// TIA Portal project "Handlings7300ip" (V15.1)

(* hardware
DEVICE "S7300/ET200M station_1"  S7-300 station
   slot 0: "Rail_0"  Rail  6ES7 390-1***0-0AA0
   slot 2: "PLC_1"  CPU 314C-2 PN/DP  6ES7 314-6EH04-0AB0  V3.3
      slot 2: "PROFINET interface_1"  PN-IO
         slot 1: "Port_1"  Port
         slot 2: "Port_2"  Port
      slot 5: "DI 24/DO 16_1"  DI24/DO16
      slot 6: "AI 5/AO 2_1"  AI5/AO2
      slot 7: "Count_1"  Counter
      slot 8: "Positioning_1"  Positioning
   slot 4: "DO 8x24VDC/0.5A_1"  DO8 x 24VDC / 0.5A  6ES7 322-8BF00-0AB0
*)

// ===== PLC "PLC_1"  CPU 314C-2 PN/DP =====

VAR_GLOBAL   // PLC tag table "Default tag table"
   "Auto" AT %I0.0 : Bool;
   "Manua" AT %I0.1 : Bool;
   "S1_Nipper_out" AT %I0.2 : Bool;
   "S2_Nipper_in" AT %I0.3 : Bool;
   "S3_Nipper_off" AT %I0.4 : Bool;
   "S5_Nipper_up" AT %I0.5 : Bool;
   "S6_Nipper_down" AT %I0.6 : Bool;
   "Start" AT %I1.0 : Bool;
   "Stop" AT %I1.1 : Bool;
   "Reset" AT %I1.2 : Bool;
   "A1" AT %I1.3 : Bool;
   "A2" AT %I1.4 : Bool;
   "B1" AT %I1.5 : Bool;
   "B2" AT %I2.0 : Bool;
   "C1" AT %I2.1 : Bool;
   "C2" AT %I2.2 : Bool;
   "1Y2" AT %Q0.0 : Bool;
   "1Y1" AT %Q0.1 : Bool;
   "2Y1" AT %Q0.2 : Bool;
   "M+" AT %Q0.3 : Bool;
   "M-" AT %Q0.4 : Bool;
   "H_Auto" AT %Q0.5 : Bool;
   "H_Manual" AT %Q0.6 : Bool;
END_VAR

DATA_BLOCK "Master_DB"   // DB1
{ S7_Optimized_Access := 'FALSE' }
VERSION : 0.1
// stored: InstanceOfName Master
"Master"
BEGIN
END_DATA_BLOCK

DATA_BLOCK "Auto_Mode_DB"   // DB2
{ S7_Optimized_Access := 'FALSE' }
VERSION : 0.1
// stored: InstanceOfName Auto_Mode
"Auto_Mode"
BEGIN
END_DATA_BLOCK

DATA_BLOCK "Output_DB"   // DB3
{ S7_Optimized_Access := 'FALSE' }
VERSION : 0.1
// stored: InstanceOfName Output
"Output"
BEGIN
END_DATA_BLOCK

DATA_BLOCK "Manual_Mode_DB"   // DB4
{ S7_Optimized_Access := 'FALSE' }
VERSION : 0.1
// stored: InstanceOfName Manual_Mode
"Manual_Mode"
BEGIN
END_DATA_BLOCK

DATA_BLOCK "Resets_DB"   // DB5
{ S7_Optimized_Access := 'FALSE' }
VERSION : 0.1
// stored: InstanceOfName Resets
"Resets"
BEGIN
END_DATA_BLOCK

FUNCTION_BLOCK "Master"   // FB1, FBD
{ S7_Optimized_Access := 'FALSE' }
VERSION : 0.1
   VAR_INPUT
      Auto : Bool;
      Manual : Bool;
      Start : Bool;
      Stop : Bool;
      Reset : Bool;
      S1 : Bool;
      S2 : Bool;
      S3 : Bool;
      S5 : Bool;
      S6 : Bool;
      "G_Reset.X200" : Bool;
      "G_Reset.X201" : Bool;
   END_VAR
   VAR_OUTPUT
      H_Auto : Bool;
      H_Manual : Bool;
      G_Auto_mode : Bool;
      G_Manual_mode : Bool;
   END_VAR
   VAR
      X0 : Bool;
      X1 : Bool;
      X2 : Bool;
      X3 : Bool;
   END_VAR
BEGIN

REGION Network 1
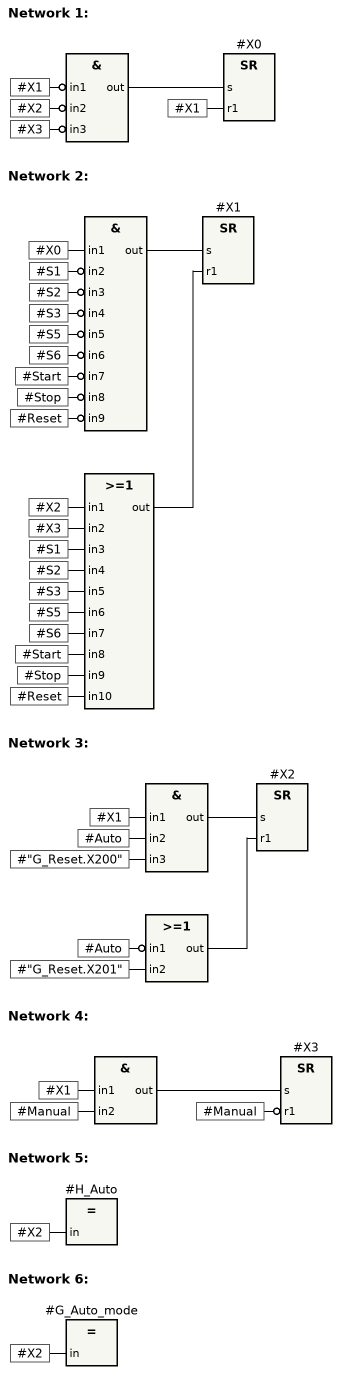
   IF NOT #X1 AND NOT #X2 AND NOT #X3 THEN
       #X0 := TRUE;   // SR flip-flop
   END_IF;
   IF #X1 THEN #X0 := FALSE; END_IF;
END_REGION

REGION Network 2
   IF #X0 AND NOT #S1 AND NOT #S2 AND NOT #S3 AND NOT #S5 AND NOT #S6 AND NOT #Start AND NOT #Stop AND NOT #Reset THEN
       #X1 := TRUE;   // SR flip-flop
   END_IF;
   IF #X2 OR #X3 OR #S1 OR #S2 OR #S3 OR #S5 OR #S6 OR #Start OR #Stop OR #Reset THEN #X1 := FALSE; END_IF;
END_REGION

REGION Network 3
   IF #X1 AND #Auto AND #"G_Reset.X200" THEN
       #X2 := TRUE;   // SR flip-flop
   END_IF;
   IF NOT #Auto OR #"G_Reset.X201" THEN #X2 := FALSE; END_IF;
END_REGION

REGION Network 4
   IF #X1 AND #Manual THEN
       #X3 := TRUE;   // SR flip-flop
   END_IF;
   IF NOT #Manual THEN #X3 := FALSE; END_IF;
END_REGION

REGION Network 5
   #H_Auto := #X2;
END_REGION

REGION Network 6
   #G_Auto_mode := #X2;
END_REGION

REGION Network 7
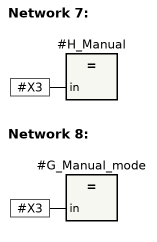
   #H_Manual := #X3;
END_REGION

REGION Network 8
   #G_Manual_mode := #X3;
END_REGION
END_FUNCTION_BLOCK

FUNCTION_BLOCK "Auto_Mode"   // FB2, FBD
{ S7_Optimized_Access := 'FALSE' }
VERSION : 0.1
   VAR_INPUT
      Auto_mode : Bool;
      Start : Bool;
      Stop : Bool;
      Reset : Bool;
      A1 : Bool;
      A2 : Bool;
      B1 : Bool;
      B2 : Bool;
      C1 : Bool;
      C2 : Bool;
   END_VAR
   VAR_OUTPUT
      Nipper_out_1Y1_A : Bool;
      Nipper_in_1Y2_A : Bool;
      Nipper_off_2Y1_A : Bool;
      Nipper_up_A : Bool;
      Nipper_down_A : Bool;
   END_VAR
   VAR
      X10 : Bool;
      X11 : Bool;
      X12 : Bool;
      X13 : Bool;
      X14 : Bool;
      X15 : Bool;
      X16 : Bool;
      X17 : Bool;
      X18 : Bool;
   END_VAR
BEGIN

REGION Network 1
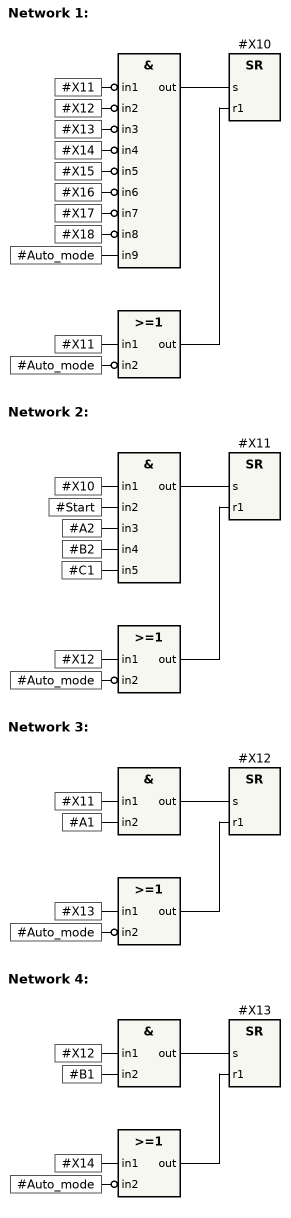
   IF NOT #X11 AND NOT #X12 AND NOT #X13 AND NOT #X14 AND NOT #X15 AND NOT #X16 AND NOT #X17 AND NOT #X18 AND #Auto_mode THEN
       #X10 := TRUE;   // SR flip-flop
   END_IF;
   IF #X11 OR NOT #Auto_mode THEN #X10 := FALSE; END_IF;
END_REGION

REGION Network 2
   IF #X10 AND #Start AND #A2 AND #B2 AND #C1 THEN
       #X11 := TRUE;   // SR flip-flop
   END_IF;
   IF #X12 OR NOT #Auto_mode THEN #X11 := FALSE; END_IF;
END_REGION

REGION Network 3
   IF #X11 AND #A1 THEN
       #X12 := TRUE;   // SR flip-flop
   END_IF;
   IF #X13 OR NOT #Auto_mode THEN #X12 := FALSE; END_IF;
END_REGION

REGION Network 4
   IF #X12 AND #B1 THEN
       #X13 := TRUE;   // SR flip-flop
   END_IF;
   IF #X14 OR NOT #Auto_mode THEN #X13 := FALSE; END_IF;
END_REGION

REGION Network 5
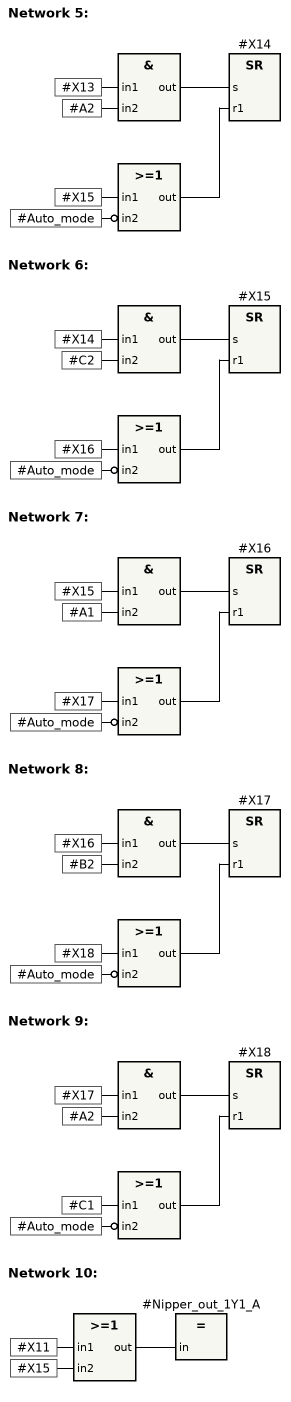
   IF #X13 AND #A2 THEN
       #X14 := TRUE;   // SR flip-flop
   END_IF;
   IF #X15 OR NOT #Auto_mode THEN #X14 := FALSE; END_IF;
END_REGION

REGION Network 6
   IF #X14 AND #C2 THEN
       #X15 := TRUE;   // SR flip-flop
   END_IF;
   IF #X16 OR NOT #Auto_mode THEN #X15 := FALSE; END_IF;
END_REGION

REGION Network 7
   IF #X15 AND #A1 THEN
       #X16 := TRUE;   // SR flip-flop
   END_IF;
   IF #X17 OR NOT #Auto_mode THEN #X16 := FALSE; END_IF;
END_REGION

REGION Network 8
   IF #X16 AND #B2 THEN
       #X17 := TRUE;   // SR flip-flop
   END_IF;
   IF #X18 OR NOT #Auto_mode THEN #X17 := FALSE; END_IF;
END_REGION

REGION Network 9
   IF #X17 AND #A2 THEN
       #X18 := TRUE;   // SR flip-flop
   END_IF;
   IF #C1 OR NOT #Auto_mode THEN #X18 := FALSE; END_IF;
END_REGION

REGION Network 10
   #Nipper_out_1Y1_A := #X11 OR #X15;
END_REGION

REGION Network 11
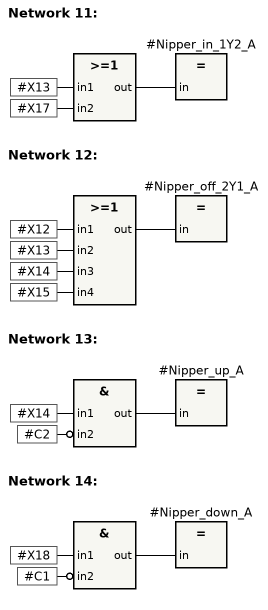
   #Nipper_in_1Y2_A := #X13 OR #X17;
END_REGION

REGION Network 12
   #Nipper_off_2Y1_A := #X12 OR #X13 OR #X14 OR #X15;
END_REGION

REGION Network 13
   #Nipper_up_A := #X14 AND NOT #C2;
END_REGION

REGION Network 14
   #Nipper_down_A := #X18 AND NOT #C1;
END_REGION
END_FUNCTION_BLOCK

FUNCTION_BLOCK "Output"   // FB3, FBD
{ S7_Optimized_Access := 'FALSE' }
VERSION : 0.1
   VAR_INPUT
      Nipper_out_1Y1_M : Bool;
      Nipper_in_1Y2_M : Bool;
      Nipper_off_2Y1_M : Bool;
      Nipper_up_M : Bool;
      Nipper_down_M : Bool;
      Nipper_out_1Y1_A : Bool;
      Nipper_in_1Y2_A : Bool;
      Nipper_off_2Y1_A : Bool;
      Nipper_up_A : Bool;
      Nipper_down_A : Bool;
      Nipper_in_1Y2_r : Bool;
      Nipper_off_2Y1_r : Bool;
      Nipper_down_r : Bool;
   END_VAR
   VAR_OUTPUT
      Nipper_out_1Y1 : Bool;
      Nipper_in_1Y2 : Bool;
      Nipper_off_2Y1 : Bool;
      Nipper_up : Bool;
      Nipper_down : Bool;
   END_VAR
BEGIN

REGION Network 1
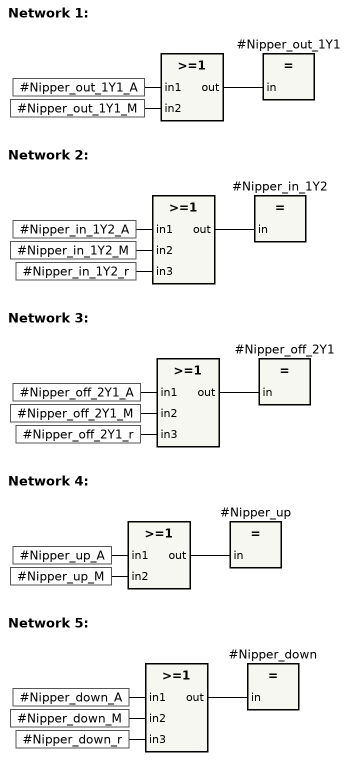
   #Nipper_out_1Y1 := #Nipper_out_1Y1_A OR #Nipper_out_1Y1_M;
END_REGION

REGION Network 2
   #Nipper_in_1Y2 := #Nipper_in_1Y2_A OR #Nipper_in_1Y2_M OR #Nipper_in_1Y2_r;
END_REGION

REGION Network 3
   #Nipper_off_2Y1 := #Nipper_off_2Y1_A OR #Nipper_off_2Y1_M OR #Nipper_off_2Y1_r;
END_REGION

REGION Network 4
   #Nipper_up := #Nipper_up_A OR #Nipper_up_M;
END_REGION

REGION Network 5
   #Nipper_down := #Nipper_down_A OR #Nipper_down_M OR #Nipper_down_r;
END_REGION
END_FUNCTION_BLOCK

FUNCTION_BLOCK "Manual_Mode"   // FB4, FBD
{ S7_Optimized_Access := 'FALSE' }
VERSION : 0.1
   VAR_INPUT
      G_Manual_mode : Bool;
      Manual : Bool;
      S1 : Bool;
      S2 : Bool;
      S3 : Bool;
      S5 : Bool;
      S6 : Bool;
      A1 : Bool;
      A2 : Bool;
      B1 : Bool;
      B2 : Bool;
      C1 : Bool;
      C2 : Bool;
   END_VAR
   VAR_OUTPUT
      Nipper_out_1Y1_M : Bool;
      Nipper_in_1Y2_M : Bool;
      Nipper_off_2Y1_M : Bool;
      Nipper_up_M : Bool;
      Nipper_down_M : Bool;
   END_VAR
   VAR
      X100 : Bool;
      X101 : Bool;
   END_VAR
BEGIN

REGION Network 1
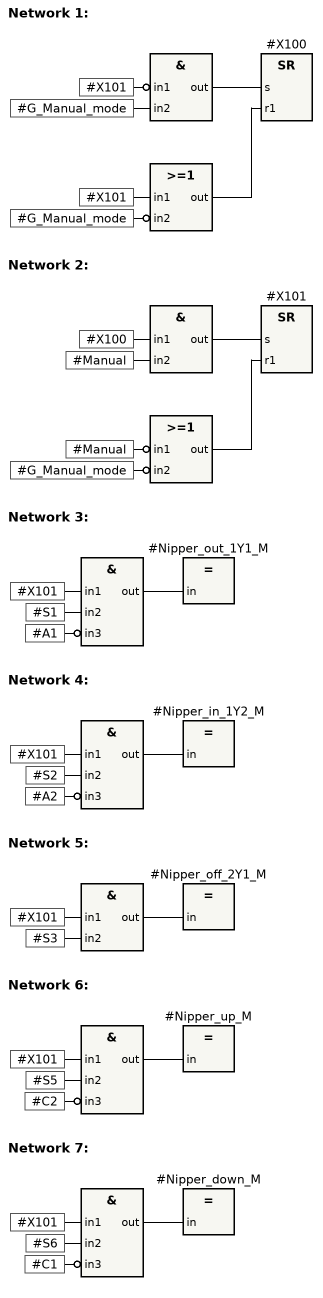
   IF NOT #X101 AND #G_Manual_mode THEN
       #X100 := TRUE;   // SR flip-flop
   END_IF;
   IF #X101 OR NOT #G_Manual_mode THEN #X100 := FALSE; END_IF;
END_REGION

REGION Network 2
   IF #X100 AND #Manual THEN
       #X101 := TRUE;   // SR flip-flop
   END_IF;
   IF NOT #Manual OR NOT #G_Manual_mode THEN #X101 := FALSE; END_IF;
END_REGION

REGION Network 3
   #Nipper_out_1Y1_M := #X101 AND #S1 AND NOT #A1;
END_REGION

REGION Network 4
   #Nipper_in_1Y2_M := #X101 AND #S2 AND NOT #A2;
END_REGION

REGION Network 5
   #Nipper_off_2Y1_M := #X101 AND #S3;
END_REGION

REGION Network 6
   #Nipper_up_M := #X101 AND #S5 AND NOT #C2;
END_REGION

REGION Network 7
   #Nipper_down_M := #X101 AND #S6 AND NOT #C1;
END_REGION
END_FUNCTION_BLOCK

FUNCTION_BLOCK "Resets"   // FB5, FBD
{ S7_Optimized_Access := 'FALSE' }
VERSION : 0.1
   VAR_INPUT
      Reset : Bool;
      Stop : Bool;
      Auto : Bool;
      A2 : Bool;
      B1 : Bool;
      B2 : Bool;
      C1 : Bool;
   END_VAR
   VAR_OUTPUT
      Nipper_in_1Y2_r : Bool;
      Nipper_off_2Y1_r : Bool;
      Nipper_down_r : Bool;
   END_VAR
   VAR
      X200 : Bool;
      X201 : Bool;
      X202 : Bool;
      X203 : Bool;
   END_VAR
BEGIN

REGION Network 1
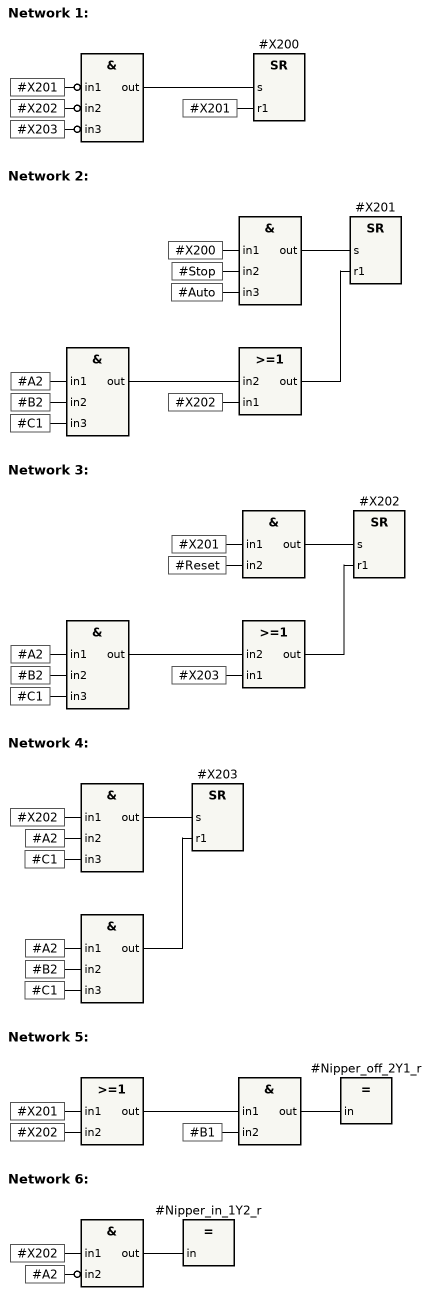
   IF NOT #X201 AND NOT #X202 AND NOT #X203 THEN
       #X200 := TRUE;   // SR flip-flop
   END_IF;
   IF #X201 THEN #X200 := FALSE; END_IF;
END_REGION

REGION Network 2
   IF #X200 AND #Stop AND #Auto THEN
       #X201 := TRUE;   // SR flip-flop
   END_IF;
   IF (#A2 AND #B2 AND #C1) OR #X202 THEN #X201 := FALSE; END_IF;
END_REGION

REGION Network 3
   IF #X201 AND #Reset THEN
       #X202 := TRUE;   // SR flip-flop
   END_IF;
   IF (#A2 AND #B2 AND #C1) OR #X203 THEN #X202 := FALSE; END_IF;
END_REGION

REGION Network 4
   IF #X202 AND #A2 AND #C1 THEN
       #X203 := TRUE;   // SR flip-flop
   END_IF;
   IF #A2 AND #B2 AND #C1 THEN #X203 := FALSE; END_IF;
END_REGION

REGION Network 5
   #Nipper_off_2Y1_r := (#X201 OR #X202) AND #B1;
END_REGION

REGION Network 6
   #Nipper_in_1Y2_r := #X202 AND NOT #A2;
END_REGION

REGION Network 7
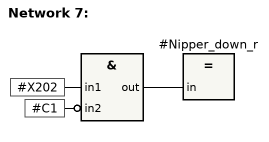
   #Nipper_down_r := #X202 AND NOT #C1;
END_REGION
END_FUNCTION_BLOCK

ORGANIZATION_BLOCK "Main"   // OB1, FBD
TITLE = "Main Program Sweep (Cycle)"
{ S7_Optimized_Access := 'FALSE' }
VERSION : 0.1
   VAR_TEMP
      OB1_EV_CLASS : Byte;   // Bits 0-3 = 1 (Coming event), Bits 4-7 = 1 (Event class 1)
      OB1_SCAN_1 : Byte;   // 1 (Cold restart scan 1 of OB 1), 3 (Scan 2-n of OB 1)
      OB1_PRIORITY : Byte;   // Priority of OB Execution
      OB1_OB_NUMBR : Byte;   // 1 (Organization block 1, OB1)
      OB1_RESERVED_1 : Byte;   // Reserved for system
      OB1_RESERVED_2 : Byte;   // Reserved for system
      OB1_PREV_CYCLE : Int;   // Cycle time of previous OB1 scan (milliseconds)
      OB1_MIN_CYCLE : Int;   // Minimum cycle time of OB1 (milliseconds)
      OB1_MAX_CYCLE : Int;   // Maximum cycle time of OB1 (milliseconds)
      OB1_DATE_TIME : Date_And_Time;   // Date and time OB1 started
   END_VAR
BEGIN

REGION Network 1
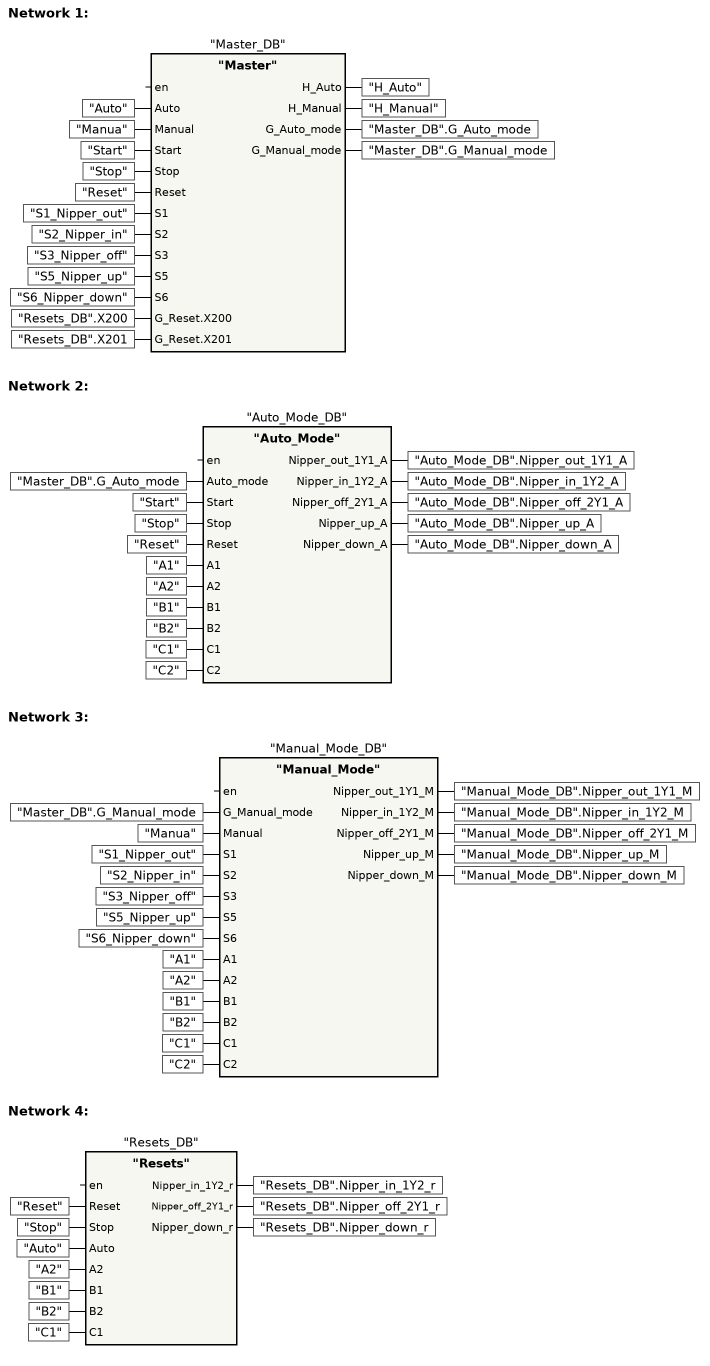
   "Master_DB"(Auto := "Auto",   // "Master"
               Manual := "Manua",
               Start := "Start",
               Stop := "Stop",
               Reset := "Reset",
               S1 := "S1_Nipper_out",
               S2 := "S2_Nipper_in",
               S3 := "S3_Nipper_off",
               S5 := "S5_Nipper_up",
               S6 := "S6_Nipper_down",
               "G_Reset.X200" := "Resets_DB".X200,
               "G_Reset.X201" := "Resets_DB".X201,
               H_Auto => "H_Auto",
               H_Manual => "H_Manual",
               G_Auto_mode => "Master_DB".G_Auto_mode,
               G_Manual_mode => "Master_DB".G_Manual_mode);
END_REGION

REGION Network 2
   "Auto_Mode_DB"(Auto_mode := "Master_DB".G_Auto_mode,   // "Auto_Mode"
                  Start := "Start",
                  Stop := "Stop",
                  Reset := "Reset",
                  A1 := "A1",
                  A2 := "A2",
                  B1 := "B1",
                  B2 := "B2",
                  C1 := "C1",
                  C2 := "C2",
                  Nipper_out_1Y1_A => "Auto_Mode_DB".Nipper_out_1Y1_A,
                  Nipper_in_1Y2_A => "Auto_Mode_DB".Nipper_in_1Y2_A,
                  Nipper_off_2Y1_A => "Auto_Mode_DB".Nipper_off_2Y1_A,
                  Nipper_up_A => "Auto_Mode_DB".Nipper_up_A,
                  Nipper_down_A => "Auto_Mode_DB".Nipper_down_A);
END_REGION

REGION Network 3
   "Manual_Mode_DB"(G_Manual_mode := "Master_DB".G_Manual_mode,   // "Manual_Mode"
                    Manual := "Manua",
                    S1 := "S1_Nipper_out",
                    S2 := "S2_Nipper_in",
                    S3 := "S3_Nipper_off",
                    S5 := "S5_Nipper_up",
                    S6 := "S6_Nipper_down",
                    A1 := "A1",
                    A2 := "A2",
                    B1 := "B1",
                    B2 := "B2",
                    C1 := "C1",
                    C2 := "C2",
                    Nipper_out_1Y1_M => "Manual_Mode_DB".Nipper_out_1Y1_M,
                    Nipper_in_1Y2_M => "Manual_Mode_DB".Nipper_in_1Y2_M,
                    Nipper_off_2Y1_M => "Manual_Mode_DB".Nipper_off_2Y1_M,
                    Nipper_up_M => "Manual_Mode_DB".Nipper_up_M,
                    Nipper_down_M => "Manual_Mode_DB".Nipper_down_M);
END_REGION

REGION Network 4
   "Resets_DB"(Reset := "Reset",   // "Resets"
               Stop := "Stop",
               Auto := "Auto",
               A2 := "A2",
               B1 := "B1",
               B2 := "B2",
               C1 := "C1",
               Nipper_in_1Y2_r => "Resets_DB".Nipper_in_1Y2_r,
               Nipper_off_2Y1_r => "Resets_DB".Nipper_off_2Y1_r,
               Nipper_down_r => "Resets_DB".Nipper_down_r);
END_REGION

REGION Network 5
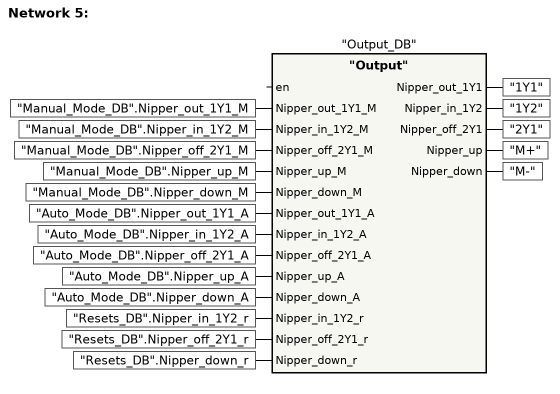
   "Output_DB"(Nipper_out_1Y1_M := "Manual_Mode_DB".Nipper_out_1Y1_M,   // "Output"
               Nipper_in_1Y2_M := "Manual_Mode_DB".Nipper_in_1Y2_M,
               Nipper_off_2Y1_M := "Manual_Mode_DB".Nipper_off_2Y1_M,
               Nipper_up_M := "Manual_Mode_DB".Nipper_up_M,
               Nipper_down_M := "Manual_Mode_DB".Nipper_down_M,
               Nipper_out_1Y1_A := "Auto_Mode_DB".Nipper_out_1Y1_A,
               Nipper_in_1Y2_A := "Auto_Mode_DB".Nipper_in_1Y2_A,
               Nipper_off_2Y1_A := "Auto_Mode_DB".Nipper_off_2Y1_A,
               Nipper_up_A := "Auto_Mode_DB".Nipper_up_A,
               Nipper_down_A := "Auto_Mode_DB".Nipper_down_A,
               Nipper_in_1Y2_r := "Resets_DB".Nipper_in_1Y2_r,
               Nipper_off_2Y1_r := "Resets_DB".Nipper_off_2Y1_r,
               Nipper_down_r := "Resets_DB".Nipper_down_r,
               Nipper_out_1Y1 => "1Y1",
               Nipper_in_1Y2 => "1Y2",
               Nipper_off_2Y1 => "2Y1",
               Nipper_up => "M+",
               Nipper_down => "M-");
END_REGION
END_ORGANIZATION_BLOCK